TYPE ST_HMI_C1_Network : 
STRUCT
	stHMI_C1_Ctrl2_PackML_Overall_Equipment_Effectiveness_OEE: ST_HMI_C1_Ctrl2_PackML_Overall_Equipment_Effectiveness_OEE;
	
	stHMI_C1_Ctrl1_Pie_Chart: ST_HMI_C1_Ctrl1_Pie_Chart;
	
	stHMI_C1_Ctrl3_Threshold_Classifier_1Ch: ST_HMI_C1_Ctrl3_Threshold_Classifier_1Ch;
	
	stHMI_C1_Ctrl4_Preventive_Maintenance_Lifetime_Analysis: ST_HMI_C1_Ctrl4_Preventive_Maintenance_Lifetime_Analysis;
	
	fN1_N1_fInput_01: LREAL;
	fN1_N1_fPlastic_Count: LREAL;
END_STRUCT
END_TYPE

(* stored: DUT ST_HMI_C1_Network: Id 07d25048-0870-4f49-b2c1-510a2396ffc0 *)
